FUNCTION_BLOCK timers_ex03
VAR_INPUT
	stand			: Switch_2P;
END_VAR
VAR_OUTPUT
	P1				: DigitalOutput;
END_VAR
VAR
	Timer1_ex03		: TOF;
	Timer2_ex03		: TON;
END_VAR

END_FUNCTION_BLOCK

(* stored: Version 1.1.0.1
   POU timers_ex03: Id {3cf5677d-42b2-4c0f-bcec-644d058688f1}, SpecialFunc None *)
